(* Logix 5000 project; controller EuniceF_ICA9 vendor 1 type 14 code 150 rev 37.11; software revision 37.00 *)

TASK MainTask (continuous, watchdog 500 ms) : MainProgram

MODULES
   Local : vendor 1 type 14 code 150 (Compact 0, rev 37.11)
      Discrete_IO : Embedded (Compact 1, rev 3.1, Output RPI 20 ms)
      Analog_IO : Embedded (Compact 2, rev 1.1, Output RPI 80 ms)
      Counters : Embedded (Compact 3, rev 1.1, Output RPI 20 ms)
END_MODULES

VAR_GLOBAL   (* controller tags *)
   CONVEYOR : ALIAS FOR Local:1:O.Data.3;
   HORN : ALIAS FOR Local:1:O.Data.2;
   RUNNING : ALIAS FOR Local:1:O.Data.0;
   RUNNING1 : ALIAS FOR Local:1:O.Data.1;
   START : ALIAS FOR Local:1:I.Data.11;
   STOP : ALIAS FOR Local:1:I.Data.8;
   Timer1 : TIMER := (PRE := 10000);
   TIMER2 : TIMER := (PRE := 4000);
END_VAR

PROGRAM MainProgram   (* main routine MainRoutine *)

ROUTINE MainRoutine   (* ladder *)
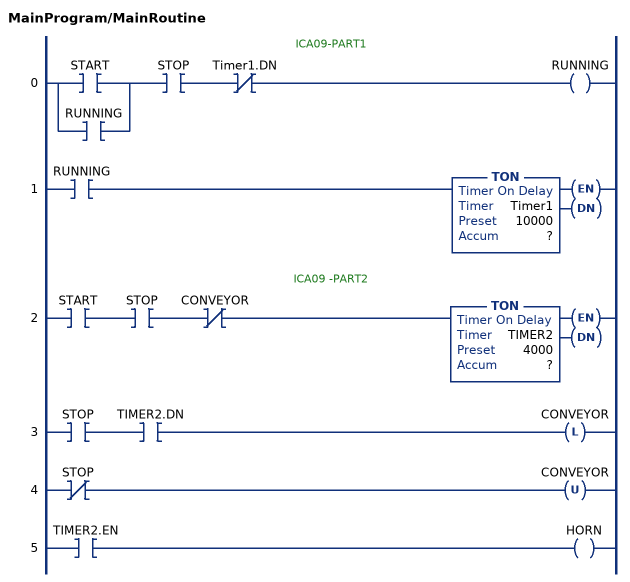
   // ICA09-PART1
   0: [XIC(START) ,XIC(RUNNING) ]XIC(STOP)XIO(Timer1.DN)OTE(RUNNING);
   1: XIC(RUNNING)TON(Timer1,?,?);
   // ICA09 -PART2
   2: XIC(START)XIC(STOP)XIO(CONVEYOR)TON(TIMER2,?,?);
   3: XIC(STOP)XIC(TIMER2.DN)OTL(CONVEYOR);
   4: XIO(STOP)OTU(CONVEYOR);
   5: XIC(TIMER2.EN)OTE(HORN);
END_ROUTINE
END_PROGRAM
